// TIA Portal project "SOMATIVA2_Ryan_yuri2024" (V17)
// HARDWARE PADRAO CLP, INTERFACES E IHM

(* hardware
DEVICE "S7-1500/ET200MP station_1"  S7-1500 station
   slot 0: "Rail_0"  Rack  6ES7 590-1***0-0AA0
   slot 1: "PLC_1"  CPU 1516-3 PN/DP  6ES7 516-3AN01-0AB0  V2.9
      slot 3: "CPU display_1"  6ES7591-1BA00-0AA0
      slot 32768: "PROFINET interface_1"  X1
      slot 33024: "PROFINET interface_2"  X2
      slot 33280: "DP interface_1"  X3
      slot 34817: "Virtual CP interface port_1"  Virtual CP interface port  Virtual CP interface port
   slot 2: "DI 32x24VDC HF_1"  DI 32x24VDC HF  6ES7 521-1BL00-0AB0  V2.1
   slot 3: "DQ 32x24VDC/0.5A HF_1"  DQ 32x24VDC/0.5A HF  6ES7 522-1BL01-0AB0  V1.0
   slot 4: "AI 8xU/I/RTD/TC ST_1"  AI 8xU/I/RTD/TC ST  6ES7 531-7KF00-0AB0  V2.0
   slot 5: "AQ 4xU/I ST_1"  AQ 4xU/I ST  6ES7 532-5HD00-0AB0  V2.0
DEVICE "HMI_1"  KTP700 Basic PN
   slot 0: "HMI_1"  KTP700 Basic PN  6AV2 123-2GB03-0AX0  14.0.1.0
   slot 1: "HMI_RT_1"  KTP700 Basic PN  6AV2 123-2GB03-0AX0  14.0.1.0
   slot 5: "HMI_1.IE_CP_1"  PROFINET Interface  14.0.1.0
      slot 1: "PROFINET Interface_1"  PROFINET Interface
         slot 1: "Port_1"  Port
*)

// ===== PLC "PLC_1"  CPU 1516-3 PN/DP =====

VAR_GLOBAL   // PLC tag table "Default tag table"
   "Clock_Byte" AT %MB100 : Byte;
   "Clock_10Hz" AT %M100.0 : Bool;
   "Clock_5Hz" AT %M100.1 : Bool;
   "Clock_2.5Hz" AT %M100.2 : Bool;
   "Clock_2Hz" AT %M100.3 : Bool;
   "Clock_1.25Hz" AT %M100.4 : Bool;
   "Clock_1Hz" AT %M100.5 : Bool;
   "Clock_0.625Hz" AT %M100.6 : Bool;
   "Clock_0.5Hz" AT %M100.7 : Bool;
END_VAR

VAR_GLOBAL   // PLC tag table "entradas_fisicas"
   "on" AT %I1.1 : Bool;
   "off" AT %I1.2 : Bool;
   "canal_0_300" AT %IW6 : Int;
   "eme" AT %I1.3 : Bool;
   "AA" AT %I0.0 : Bool;
   "RA" AT %I0.1 : Bool;
   "AB" AT %I0.2 : Bool;
   "RB" AT %I0.3 : Bool;
   "AC" AT %I0.4 : Bool;
   "RC" AT %I0.5 : Bool;
END_VAR

VAR_GLOBAL   // PLC tag table "saidas_fisicas"
   "sinVD" AT %Q1.1 : Bool;
   "sinVM" AT %Q1.3 : Bool;
   "canal_0_400" AT %QW4 : Int;
   "sinAma" AT %Q1.2 : Bool;
   "sinAzul" AT %Q1.0 : Bool;
   "helice" AT %M1.1 : Bool;
   "A" AT %Q0.0 : Bool;
   "B" AT %Q0.1 : Bool;
   "C" AT %Q0.2 : Bool;
   "V" AT %Q0.3 : Bool;
   "timer0" AT %Q0.4 : Bool;
   "timer1" AT %Q0.5 : Bool;
   "sinal" AT %Q0.7 : Bool;
END_VAR

DATA_BLOCK "Data_block_1"   // DB1
{ S7_Optimized_Access := 'TRUE' }
VERSION : 0.1
   VAR
      status : String;
      sinal : Bool;
      estado : Int := 0;
      tensaoMedida_300 : Real;
      tensaoDesejada_400 : Real;
      tela : Bool;
      ihmOn : Bool;
      ihmOff : Bool;
      leitura_300 : Real;
      escrita_400 : Real;
      trocarTelas : Array[0..3] of Int;
      scanEme : Bool;
   END_VAR
BEGIN
END_DATA_BLOCK

DATA_BLOCK "alarmes"   // DB2
{ S7_Optimized_Access := 'TRUE' }
VERSION : 0.1
   VAR
      msg : Word;
   END_VAR
BEGIN
END_DATA_BLOCK

// folder: System blocks/Program resources

DATA_BLOCK "tmr0"   // DB3
{ S7_Optimized_Access := 'TRUE' }
AUTHOR : Simatic
FAMILY : IEC
NAME : IEC_TMR
VERSION : 1.0
// stored: InstanceOfName IEC_TIMER
"IEC_TIMER"
BEGIN
END_DATA_BLOCK

DATA_BLOCK "tmr1"   // DB4
{ S7_Optimized_Access := 'TRUE' }
AUTHOR : Simatic
FAMILY : IEC
NAME : IEC_TMR
VERSION : 1.0
// stored: InstanceOfName IEC_TIMER
"IEC_TIMER"
BEGIN
END_DATA_BLOCK

// folder: (top level)

FUNCTION "trocarTelas" : Void   // FC1, LAD
{ S7_Optimized_Access := 'TRUE' }
VERSION : 0.1
   VAR_TEMP   // added for the SCL form of the ladder/FBD networks
      _w1 : Bool;
   END_VAR
BEGIN

REGION Network 1: COMANDO PRA TOCAR TELA QUANDO A EMERGÊNCIA
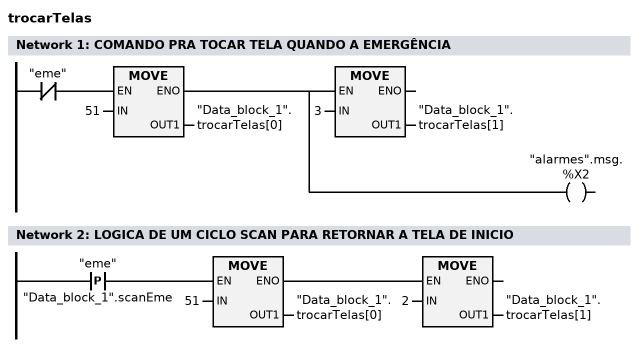
   RUNG wire#powerrail
      I_Contact( "eme" )
      Move(in := 51, out1 => "Data_block_1".trocarTelas[0])
      wire#w1
      Move(in := 3, out1 => "Data_block_1".trocarTelas[1])
   END_RUNG
   RUNG wire#w1
      Coil( "alarmes".msg.%X2 )
   END_RUNG
   // the same network as SCL:
   IF NOT "eme" THEN
       "Data_block_1".trocarTelas[0] := 51;
       "Data_block_1".trocarTelas[1] := 3;
   END_IF;
   "alarmes".msg.%X2 := NOT "eme";
END_REGION

REGION Network 2: LOGICA DE UM CICLO SCAN PARA RETORNAR A TELA DE INICIO
   RUNG wire#powerrail
      P_Contact(operand := "eme", bit := "Data_block_1".scanEme)
      Move(in := 51, out1 => "Data_block_1".trocarTelas[0])
      Move(in := 2, out1 => "Data_block_1".trocarTelas[1])
   END_RUNG
   // the same network as SCL:
   #_w1 := "eme" AND NOT "Data_block_1".scanEme;   // rising edge of "eme"
   "Data_block_1".scanEme := "eme";
   IF #_w1 THEN
       "Data_block_1".trocarTelas[0] := 51;
       "Data_block_1".trocarTelas[1] := 2;
   END_IF;
END_REGION
END_FUNCTION

ORGANIZATION_BLOCK "Main"   // OB1, LAD, ProgramCycle
TITLE = "Main Program Sweep (Cycle)"
{ S7_Optimized_Access := 'TRUE' }
VERSION : 0.1
   VAR_INPUT
      Initial_Call : Bool;   // Initial call of this OB
      Remanence : Bool;   // =True, if remanent data are available
   END_VAR
   VAR_TEMP   // added for the SCL form of the ladder/FBD networks
      _w1 : Bool;
   END_VAR
BEGIN

REGION Network 1
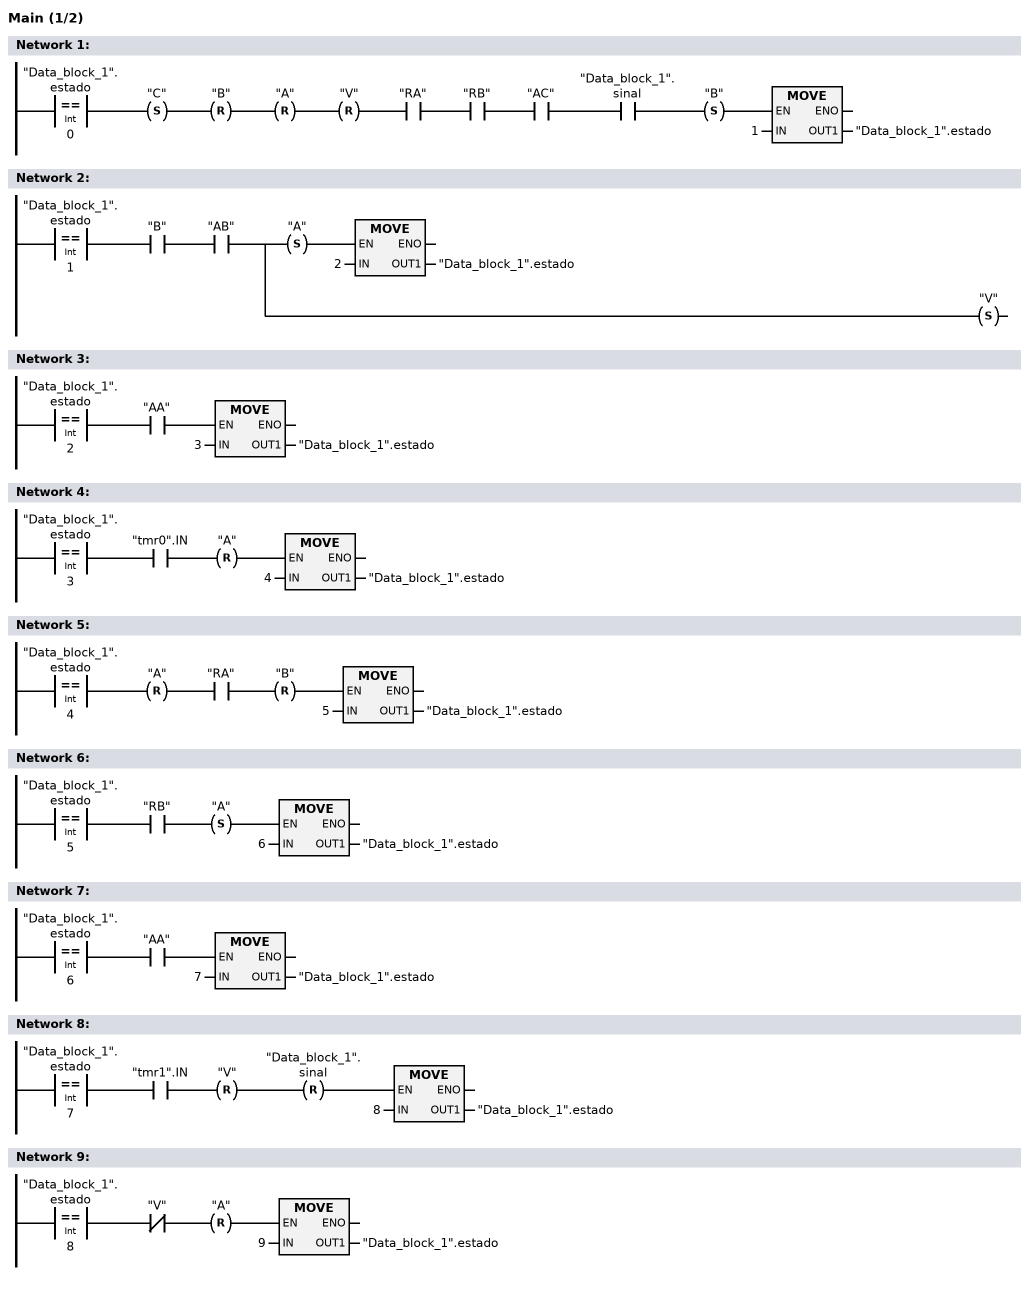
   RUNG wire#powerrail
      { S7_Templates := "SrcType := Int" } EQ_Contact(in1 := "Data_block_1".estado, in2 := 0)
      S_Coil( "C" )
      R_Coil( "B" )
      R_Coil( "A" )
      R_Coil( "V" )
      Contact( "RA" )
      Contact( "RB" )
      Contact( "AC" )
      Contact( "Data_block_1".sinal )
      S_Coil( "B" )
      Move(in := 1, out1 => "Data_block_1".estado)
   END_RUNG
   // the same network as SCL:
   #_w1 := "Data_block_1".estado = 0;
   IF #_w1 THEN
       "C" := TRUE;
       "B" := FALSE;
       "A" := FALSE;
       "V" := FALSE;
   END_IF;
   IF #_w1 AND "RA" AND "RB" AND "AC" AND "Data_block_1".sinal THEN
       "B" := TRUE;
       "Data_block_1".estado := 1;
   END_IF;
END_REGION

REGION Network 2
   RUNG wire#powerrail
      { S7_Templates := "SrcType := Int" } EQ_Contact(in1 := "Data_block_1".estado, in2 := 1)
      Contact( "B" )
      Contact( "AB" )
      wire#w1
      S_Coil( "A" )
      Move(in := 2, out1 => "Data_block_1".estado)
   END_RUNG
   RUNG wire#w1
      S_Coil( "V" )
   END_RUNG
   // the same network as SCL:
   IF ("Data_block_1".estado = 1) AND "B" AND "AB" THEN "A" := TRUE; END_IF;
   #_w1 := ("Data_block_1".estado = 1) AND "B" AND "AB";
   IF #_w1 THEN
       "Data_block_1".estado := 2;
       "V" := TRUE;
   END_IF;
END_REGION

REGION Network 3
   RUNG wire#powerrail
      { S7_Templates := "SrcType := Int" } EQ_Contact(in1 := "Data_block_1".estado, in2 := 2)
      Contact( "AA" )
      Move(in := 3, out1 => "Data_block_1".estado)
   END_RUNG
   // the same network as SCL:
   IF ("Data_block_1".estado = 2) AND "AA" THEN "Data_block_1".estado := 3; END_IF;
END_REGION

REGION Network 4
   RUNG wire#powerrail
      { S7_Templates := "SrcType := Int" } EQ_Contact(in1 := "Data_block_1".estado, in2 := 3)
      Contact( "tmr0".IN )
      R_Coil( "A" )
      Move(in := 4, out1 => "Data_block_1".estado)
   END_RUNG
   // the same network as SCL:
   IF ("Data_block_1".estado = 3) AND "tmr0".IN THEN
       "A" := FALSE;
       "Data_block_1".estado := 4;
   END_IF;
END_REGION

REGION Network 5
   RUNG wire#powerrail
      { S7_Templates := "SrcType := Int" } EQ_Contact(in1 := "Data_block_1".estado, in2 := 4)
      R_Coil( "A" )
      Contact( "RA" )
      R_Coil( "B" )
      Move(in := 5, out1 => "Data_block_1".estado)
   END_RUNG
   // the same network as SCL:
   #_w1 := "Data_block_1".estado = 4;
   IF #_w1 THEN "A" := FALSE; END_IF;
   IF #_w1 AND "RA" THEN
       "B" := FALSE;
       "Data_block_1".estado := 5;
   END_IF;
END_REGION

REGION Network 6
   RUNG wire#powerrail
      { S7_Templates := "SrcType := Int" } EQ_Contact(in1 := "Data_block_1".estado, in2 := 5)
      Contact( "RB" )
      S_Coil( "A" )
      Move(in := 6, out1 => "Data_block_1".estado)
   END_RUNG
   // the same network as SCL:
   IF ("Data_block_1".estado = 5) AND "RB" THEN
       "A" := TRUE;
       "Data_block_1".estado := 6;
   END_IF;
END_REGION

REGION Network 7
   RUNG wire#powerrail
      { S7_Templates := "SrcType := Int" } EQ_Contact(in1 := "Data_block_1".estado, in2 := 6)
      Contact( "AA" )
      Move(in := 7, out1 => "Data_block_1".estado)
   END_RUNG
   // the same network as SCL:
   IF ("Data_block_1".estado = 6) AND "AA" THEN "Data_block_1".estado := 7; END_IF;
END_REGION

REGION Network 8
   RUNG wire#powerrail
      { S7_Templates := "SrcType := Int" } EQ_Contact(in1 := "Data_block_1".estado, in2 := 7)
      Contact( "tmr1".IN )
      R_Coil( "V" )
      R_Coil( "Data_block_1".sinal )
      Move(in := 8, out1 => "Data_block_1".estado)
   END_RUNG
   // the same network as SCL:
   IF ("Data_block_1".estado = 7) AND "tmr1".IN THEN
       "V" := FALSE;
       "Data_block_1".sinal := FALSE;
       "Data_block_1".estado := 8;
   END_IF;
END_REGION

REGION Network 9
   RUNG wire#powerrail
      { S7_Templates := "SrcType := Int" } EQ_Contact(in1 := "Data_block_1".estado, in2 := 8)
      I_Contact( "V" )
      R_Coil( "A" )
      Move(in := 9, out1 => "Data_block_1".estado)
   END_RUNG
   // the same network as SCL:
   IF ("Data_block_1".estado = 8) AND NOT "V" THEN
       "A" := FALSE;
       "Data_block_1".estado := 9;
   END_IF;
END_REGION

REGION Network 10
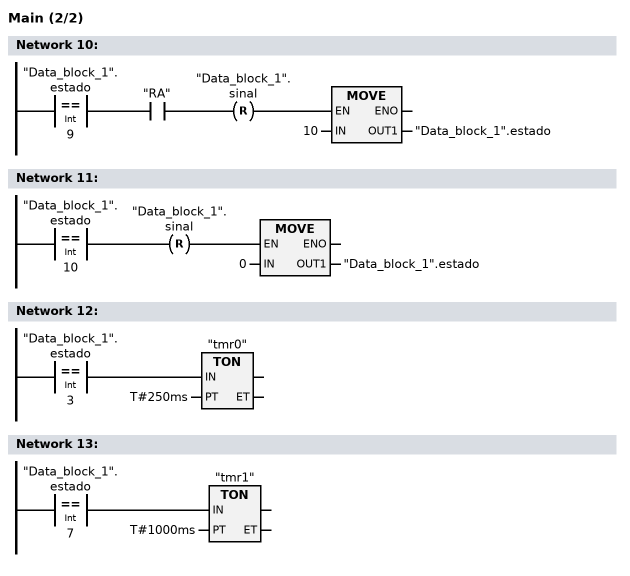
   RUNG wire#powerrail
      { S7_Templates := "SrcType := Int" } EQ_Contact(in1 := "Data_block_1".estado, in2 := 9)
      Contact( "RA" )
      R_Coil( "Data_block_1".sinal )
      Move(in := 10, out1 => "Data_block_1".estado)
   END_RUNG
   // the same network as SCL:
   IF ("Data_block_1".estado = 9) AND "RA" THEN
       "Data_block_1".sinal := FALSE;
       "Data_block_1".estado := 10;
   END_IF;
END_REGION

REGION Network 11
   RUNG wire#powerrail
      { S7_Templates := "SrcType := Int" } EQ_Contact(in1 := "Data_block_1".estado, in2 := 10)
      R_Coil( "Data_block_1".sinal )
      Move(in := 0, out1 => "Data_block_1".estado)
   END_RUNG
   // the same network as SCL:
   IF "Data_block_1".estado = 10 THEN
       "Data_block_1".sinal := FALSE;
       "Data_block_1".estado := 0;
   END_IF;
END_REGION

REGION Network 12
   "tmr0".TON(IN := "Data_block_1".estado = 3, PT := T#250ms);
END_REGION

REGION Network 13
   "tmr1".TON(IN := "Data_block_1".estado = 7, PT := T#1000ms);
END_REGION
END_ORGANIZATION_BLOCK

(* ===== HMI "HMI_RT_1" =====
system functions are stored by id; their names below are inferred from use
connection "HMI_Connection_1": ETHERNET, SMART_S7_1500_OMS

HMI tags "Default tag table"
   "sinVM" : Bool = PLC sinVM AT %Q1.3, 100 ms
   "sinVD" : Bool = PLC sinVD AT %Q1.1, 100 ms
   "Data_block_1_ihmOn" : Bool = PLC Data_block_1.ihmOn, 100 ms
   "Data_block_1_ihmOff" : Bool = PLC Data_block_1.ihmOff, 100 ms
   "Data_block_1_status" : String[254] = PLC Data_block_1.status, 100 ms
   "Data_block_1_tensaoDesejada_400" : Real = PLC Data_block_1.tensaoDesejada_400, 100 ms
   "Data_block_1_tensaoMedida_300" : Real = PLC Data_block_1.tensaoMedida_300, 100 ms
   "sinAma" : Bool = PLC sinAma AT %Q1.2, 100 ms
   "sinAzul" : Bool = PLC sinAzul AT %Q1.0, 100 ms
   "canal_0_300" : Int = PLC canal_0_300 AT %IW6, 100 ms
   "helice" : Bool = PLC helice AT %M1.1, 100 ms
   "Data_block_1_tela" : Bool = PLC Data_block_1.tela, 100 ms
   "alarmes_msg" : Word = PLC alarmes.msg, 100 ms
   "A" : Bool = PLC A AT %Q0.0, 1 s
   "B" : Bool = PLC B AT %Q0.1, 1 s
   "C" : Bool = PLC C AT %Q0.2, 1 s
   "V" : Bool = PLC V AT %Q0.3, 1 s

discrete alarms
   1: 'Motor ligado', class Warnings, trigger "alarmes_msg" bit 0
   2: 'Motor desligado', class Warnings, trigger "alarmes_msg" bit 1
   3: 'EMERGENCIA', class Errors, trigger "alarmes_msg" bit 2

analog alarms
   1: 'Tesão alta! / Alerta, nível da água acima de 9!!!', class Warnings, trigger "Data_block_1_tensaoMedida_300"
   2: 'Tesão excessiva, risco a interface / Acima de 10V, a entrada do cartão analógico corre o risco de sofrer uma pane, verifique o transdutor de temperatura urgente para identificar o seu problema. É altamente recomendável que o sistema seja desligado para uma manutenção corretiva!', class Errors, trigger "Data_block_1_tensaoMedida_300"
   3: 'EMERGENCIAAAA', class Errors, trigger "Data_block_1_tensaoMedida_300"

text list "volt": 0 '0V'; 2 '2V'; 4 '4V'; 6 '6V'; 8 '8V'; 10 '10V'

Template "Template_1" 800x480
   Button "Exit" at 714,429 size 71x50; TextOff 'Exit'; PictureOff "ExitRuntime_KTP700_Basic_PN_TR"; PictureOn "ExitRuntime_KTP700_Basic_PN_TR"
      on Release: StopRuntime(0)
   Button "Template_Button" at 614,429 size 71x50; TextOff 'Text'
   Button "Template_Button_1" at 514,429 size 71x50; TextOff 'Text'
   Button "Template_Button_2" at 414,429 size 71x50; TextOff 'Text'
   Button "Template_Button_3" at 314,429 size 71x50; TextOff 'Text'
   Button "Template_Button_4" at 214,429 size 71x50; TextOff 'Text'
   Button "Template_Button_5" at 114,429 size 71x50; TextOff 'Text'
   Button "Start screen" at 14,429 size 71x50; TextOff 'Start screen'; PictureOff "NavigateHome_KTP700_Basic_PN_TR"; PictureOn "NavigateHome_KTP700_Basic_PN_TR"
      on Release: ActivateScreen("Root screen", 0)

screen "Root screen" 800x480, template "Template_1"
   Softkey "Softkey_F2" at 0,0 size 0x0; SoftkeyImage "Left_Arrow"
      on KeyDown: ActivateScreen("INICIO", 2)
   TextField "Text field_1" at 275,62 size 230x33; Text 'Display hidrelétrica'
   UserView "User view_1" at 458,0 size 342x53
   GraphicView "Graphic view_1" at 18,150 size 211x48; Picture "pistaoAvancado"
      Visibility <- "A"
   GraphicView "Graphic view_2" at 26,155 size 103x38; Picture "Captura_de_tela_2024-05-10_201654-removebg-preview-Photoroom (2)"
      Visibility <- "A"
   GraphicView "Graphic view_4" at 276,151 size 211x48; Picture "pistaoAvancado"
      Visibility <- "B"
   GraphicView "Graphic view_5" at 285,155 size 103x38; Picture "Captura_de_tela_2024-05-10_201654-removebg-preview-Photoroom (2)"
      Visibility <- "B"
   GraphicView "Graphic view_6" at 523,153 size 211x48; Picture "pistaoAvancado"
      Visibility <- "C"
   GraphicView "Graphic view_7" at 532,157 size 103x38; Picture "Captura_de_tela_2024-05-10_201654-removebg-preview-Photoroom (2)"
      Visibility <- "C"
   GraphicView "Graphic view_8" at 284,277 size 116x88; Picture "DESENTUPAS"
      Visibility <- "V"
   GraphicView "Graphic view_9" at 354,278 size 116x88; Picture "DESENTUPAS"
      Visibility <- "V"
   TextField "Text field_2" at 75,115 size 17x23; Text 'A'
   TextField "Text field_3" at 322,115 size 16x23; Text 'B'
   TextField "Text field_4" at 577,119 size 16x23; Text 'C'
   TextField "Text field_5" at 320,266 size 16x23; Text 'V'

screen "INICIO" 800x480
   Softkey "Softkey_F3" at 0,0 size 0x0; SoftkeyImage "projeto"; Authorization "Engenharia"
      on KeyDown: ActivateScreen("Root screen", 1)
   GraphicView "Graphic view_1" at 6,1 size 93x76; Picture "LOGO_1"
   TextField "Text field_1" at 302,17 size 252x29; Text 'SOMATIVA- Ryan e Yuri'
   Button "Button_1" at 0,85 size 110x51; TextOff 'DETALHES'
      on Press: function_b14e0dd5("Data_block_1_ihmOn", 0)
      Visibility <- "Data_block_1_tela"
   Button "Button_2" at 1,85 size 109x51; TextOff 'MINIMIZAR'
      on Press: function_b14e0dd5("Data_block_1_ihmOff", 0)
      Visibility <- "Data_block_1_tela"
   Rectangle "Rectangle_2" at 196,69 size 492x322
      Visibility <- "Data_block_1_tela"
   TextField "Text field_2" at 228,196 size 433x23; Text 'O objetivo dessa atividade somativa e escalonar um'
      Visibility <- "Data_block_1_tela"
   UserView "User view_1" at 319,419 size 342x53
   TextField "Text field_3" at 231,219 size 416x42; Text 'processo produtivo real a partir de duas células de preparação e movimento dos materiais.'
      Visibility <- "Data_block_1_tela"
   Softkey "Softkey_F8" at 0,0 size 0x0; SoftkeyImage "chave"
      on KeyDown: function_f23ef4c9()

screen "Tela_emergencia" 800x480
   GraphicView "Graphic view_1" at 185,34 size 411x299; Picture "Graphic_9"
   TextField "Text field_1" at 273,340 size 224x43; Text 'EMERGÊNCIA'

screen "AlarmesRT" 800x480
   AlarmView "Alarm view_1" at 122,63 size 600x300
   TextField "Text field_1" at 117,7 size 209x29; Text 'Alarmes tempo real'
   UserView "User view_1" at 458,0 size 342x53
   Softkey "Softkey_F1" at 0,0 size 0x0; SoftkeyImage "Left_Arrow"
      on KeyDown: ActivateScreen("INICIO", 0)

screen "AlarmesLog" 800x480
   AlarmView "Alarm view_1" at 98,67 size 600x300
   TextField "Text field_1" at 91,0 size 208x32; Text 'Alarmes histórico'
   UserView "User view_1" at 458,0 size 342x53
   Softkey "Softkey_F1" at 0,0 size 0x0; SoftkeyImage "Left_Arrow"
      on KeyDown: ActivateScreen("INICIO", 0)

screen "Screen_1" 800x480
   AlarmView "Alarm view_1" at 122,63 size 600x300
*)